// TIA Portal V19 export
FUNCTION_BLOCK "G120 Comm"   // FB5, LAD
{ S7_Optimized_Access := 'TRUE' }
// stored: MemoryReserve 100, SetENOAutomatically false
   VAR_OUTPUT
      AnalogInput : Real;   // %
   END_VAR
   VAR
      WRREC_Instance { S7_SetPoint := 'True'} : WRREC;
      RDREC_Instance { S7_SetPoint := 'True'} : RDREC;
      WriteRecord : Struct
         Static_1 { S7_SetPoint := 'True'} : "HEADER";
         Static_2 { S7_SetPoint := 'True'} : "PARAMETERADDR";
      END_STRUCT;
      ReadRecord : Struct
         data : Array[0..5] of Byte;
         Value : Real;
      END_STRUCT;
   END_VAR
   // WriteRecord.Static_1.REQ_REF := 1;
   // WriteRecord.Static_1.REQ_ID := 1;
   // WriteRecord.Static_1.AXIS := 1;
   // WriteRecord.Static_1.NO_PARAM := 1;
   // WriteRecord.Static_2.ATTRIBUTE := 16;
   // WriteRecord.Static_2.NO_ELEM := 1;
   // WriteRecord.Static_2.PARA_NO := 755;
   // WriteRecord.Static_2.SUBINDEX := 0;
   VAR_TEMP   // added for the SCL form of the ladder/FBD networks
      _w1 : Bool;
   END_VAR
BEGIN

REGION Network 1
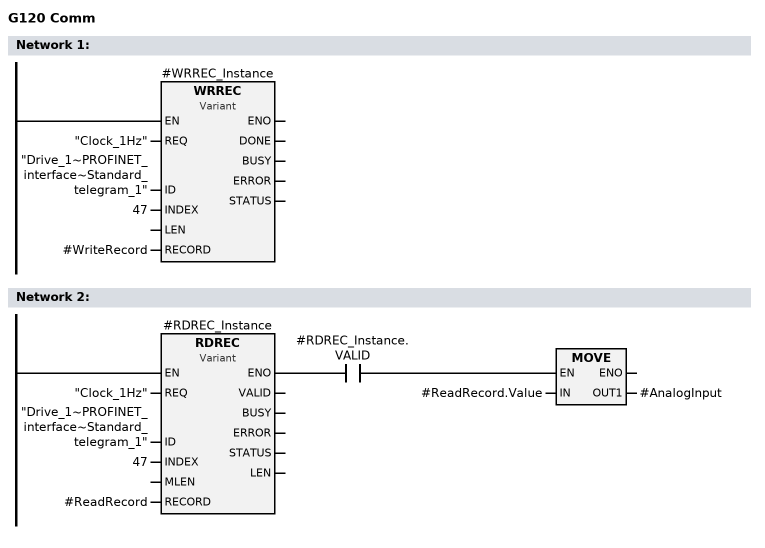
   RUNG wire#powerrail
      { S7_Templates := "[ptr_type := Variant, id_type := HW_IO, index_type := DInt, len_type := UInt]" } #WRREC_Instance.WRREC(REQ := "Clock_1Hz", ID := "Drive_1~PROFINET_interface~Standard_telegram_1", INDEX := 47, LEN :=, RECORD := #WriteRecord, DONE =>, BUSY =>, ERROR =>, STATUS =>)
   END_RUNG
   // the same network as SCL:
   #WRREC_Instance(REQ := "Clock_1Hz",   // WRREC
                   ID := "Drive_1~PROFINET_interface~Standard_telegram_1",
                   INDEX := 47,
                   RECORD := #WriteRecord);
END_REGION

REGION Network 2
   RUNG wire#powerrail
      { S7_Templates := "[ptr_type := Variant, id_type := HW_IO, index_type := DInt, len_type := UInt]" } #RDREC_Instance.RDREC(REQ := "Clock_1Hz", ID := "Drive_1~PROFINET_interface~Standard_telegram_1", INDEX := 47, MLEN :=, RECORD := #ReadRecord, VALID =>, BUSY =>, ERROR =>, STATUS =>, LEN =>)
      Contact( #RDREC_Instance.VALID )
      Move(in := #ReadRecord.Value, out1 => #AnalogInput)
   END_RUNG
   // the same network as SCL:
   #RDREC_Instance(REQ := "Clock_1Hz",   // RDREC
                   ID := "Drive_1~PROFINET_interface~Standard_telegram_1",
                   INDEX := 47,
                   RECORD := #ReadRecord,
                   ENO => #_w1);
   IF #_w1 AND #RDREC_Instance.VALID THEN #AnalogInput := #ReadRecord.Value; END_IF;
END_REGION
END_FUNCTION_BLOCK
